FUNCTION_BLOCK ABSTRACT RfidBase EXTENDS TExecution IMPLEMENTS IDevice
VAR_INPUT
END_VAR
VAR_OUTPUT
END_VAR
VAR
	{attribute 'OPC.UA.DA' := '0'}
	_name : STRING;
	{attribute 'OPC.UA.DA' := '0'}
	_deviceID : STRING;				
	{attribute 'OPC.UA.DA' := '0'}	
	_family : DeviceFamily;	
	{attribute 'OPC.UA.DA' := '0'}
	_logger : Logger;
	{attribute 'OPC.UA.DA' := '0'}
	_message : StringBuilder;
	{attribute 'OPC.UA.DA' := '0'}
	_rfidConfig : DeviceConfiguration;	
END_VAR

PROPERTY DeviceID : STRING
GET
DeviceID := _deviceID;
END_GET
SET
_deviceID := DeviceID;
END_SET
END_PROPERTY

PROPERTY Family : DeviceFamily
GET
Family := _family;
END_GET
SET
_family := Family;
END_SET
END_PROPERTY

PROPERTY Name : STRING
GET
Name := _name;
END_GET
SET
_name := Name;
END_SET
END_PROPERTY

END_FUNCTION_BLOCK

(* stored: Version 1.1.0.1, ProductVersion 3.1.4024.12
   POU RfidBase: Id {f40d3132-c9e2-485d-8c31-12b3909d48ec}, SpecialFunc None
   Property DeviceID: Id {dcfa8958-a0f7-4510-99eb-002410140fbc}
   Get Get: Id {ba14c7cd-e621-484f-b0a9-72f19ed86f27}
   Set Set: Id {7ee509bc-7fef-4498-a5a1-5940042facc8}
   Property Family: Id {e80fa4e3-aa4b-4783-8115-2e4829821ca4}
   Get Get: Id {f40ecc90-8244-43b4-95c3-b74108ca1dfa}
   Set Set: Id {eddefffc-f1f0-4563-9f30-7e251f75b51b}
   Property Name: Id {26f75eb9-4ea3-4c9e-a57e-38d1725f6b4b}
   Get Get: Id {e632df79-8426-42ce-acb7-2ec467fbed95}
   Set Set: Id {7e5a312a-bcf2-48d0-8f86-199c263d0fdb} *)
